PROGRAM MAIN
VAR
	 fbAlarm : FB_AlarmController;
END_VAR

fbAlarm();

END_PROGRAM

(* stored: Version 1.1.0.1, ProductVersion 3.1.4024.16
   POU MAIN: Id {290377bf-b4e5-4a72-86a7-d35d66667e63}, SpecialFunc None *)
